// SIMATIC S7-200 project (STEP 7-Micro/WIN), CPU 221 REL 01.10

SYMBOL_TABLE USER1
S1               I0.0     // DEM TANG
S2               I0.1     // DEM GIAM
Y                Q0.0     // DEN BAO DAY
S3               Q0.2     // RESET
END_SYMBOL_TABLE

ORGANIZATION_BLOCK MAIN:OB1
TITLE=PROGRAM COMMENTS
BEGIN
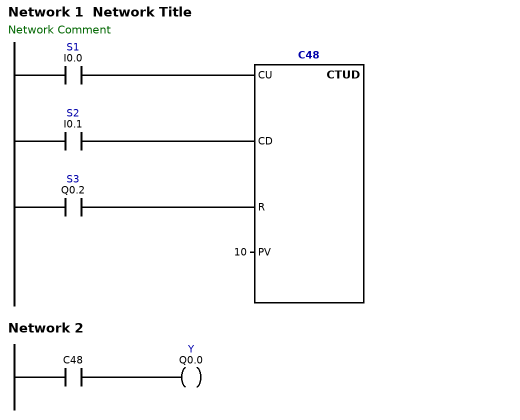
Network 1 // Network Title
// Network Comment
LD     S1:I0.0
LD     S2:I0.1
LD     S3:Q0.2
CTUD   C48, 10
Network 2
LD     C48
=      Y:Q0.0
END_ORGANIZATION_BLOCK
